// TIA Portal V20 export
TYPE "LKinCtrl_PointEditor_typeUndoBuffer"
// stored: Access Published
   STRUCT
      index { ExternalAccessible := 'False'; ExternalVisible := 'False'; ExternalWritable := 'False'} : Int;   // current index in the buffer.
      stepsRedo { ExternalAccessible := 'False'; ExternalVisible := 'False'; ExternalWritable := 'False'} : Int;   // possible steps for redo.
      stepsUndo { ExternalAccessible := 'False'; ExternalVisible := 'False'; ExternalWritable := 'False'} : Int;   // possible steps for undo.
      entries { ExternalAccessible := 'False'; ExternalVisible := 'False'; ExternalWritable := 'False'} : Array[0.."LKINCTRL_NO_OF_POINT_UNDOS_POINT_EDITOR"] of Struct   // entries in buffer.
         coordinateSystem : DInt;
         point : "LKinCtrl_PointEditor_typePoint";
      END_STRUCT;
   END_STRUCT;
END_TYPE
